// A CoE transfer that an I_CoeTransferScheduler services each cycle while Busy is TRUE.
INTERFACE I_CoeTransfer EXTENDS I_Cyclic, I_TaskResult

END_INTERFACE

(* stored: Version 1.1.0.1, ProductVersion 3.1.4026.18
   Itf I_CoeTransfer: Id {ddf158f5-3687-4c26-8621-5d7379b7d5c3} *)
